Fanuc KAREL source: kc00004.KL

-- PROVISIONAL review KL for V940-1; original PC SHA256 b28ee204621b1c3c830ec8505e500cc4c40f5254ab9ed6aa19b091163028b9ff
-- Incomplete behavior may be omitted. Consult companion uncertainty JSON. Do not deploy.
PROGRAM KC00004
%NOLOCKGROUP
BEGIN
  -- V9_ZERO_TABLE_METADATA_HINT layout=0002_ascii; no indexed target words; source/name/runtime held
  -- UNRESOLVED_PC offsets 5-35; opcodes 27,22,22,22,2A,22,31
  -- UNRESOLVED_PC offsets 40-44; opcodes 7F
END KC00004
